{attribute 'OPC.UA.DA.StructuredType' := '1'}
TYPE ST_TestSystemState :
STRUCT
	//general information
	bOperational				: BOOL;
END_STRUCT
END_TYPE

(* stored: Version 1.1.0.1, ProductVersion 3.1.4024.9
   DUT ST_TestSystemState: Id {48e0cba5-b086-4590-99b5-594598371795} *)
